Staubli VAL3: pulse.pgx

public program pulse(dio x_dDio, num x_nLength)
begin

  //generates a pulse of x_nLength for the output x_dDio

  if taskStatus("pulse_"+toString("",nPulseCount))==-1
    taskCreate "pulse_"+toString("",nPulseCount),10,exePulse(x_dDio,x_nLength)
    nPulseCount=nPulseCount+1
    if nPulseCount>nMaxTask
      nPulseCount=0
    endIf
  else
    logMsg("libSignals/pulse->can't create the task!")
  endIf

end
